FUNCTION_BLOCK  FB_NCU_Base
//////////////////
// NCU Function 
//////////////////
VAR_INPUT PERSISTENT
	// Parameters of the Object (instance/model specific) 
	ParamIPAddress				: STRING := '192.168.1.1' ; // IP 
	ParamTcpPort				: UINT		:= 502;
	ParamTimeOut				: TIME := T#10S ; 
	ParamClockReadTime			: TIME := T#1S ; 
	
	ParamClockWriteTime			: TIME := T#1S ; 	
	
	ParamUnitID 				: BYTE:=1; 					// (NA)   SMA Modbus Unit ID.
	ParamNbTracker				: BYTE ; 					// Number of tracker behind the 
	ParamNCUNum					: INT ; 					// Numerous of TCU 
	                                                		
	ParamTempoComAlarm			: TIME 			 ; 			// (s) Config : Tempo to detect LOC Alarm	

END_VAR

VAR_INPUT 
	//Child objects
	IN_CmdReset_L							: BOOL;				// (NA) External Reset Command	
    IN_CmdToggleRead						: BOOL;
    IN_CmdToggleWrite						: BOOL;
END_VAR


VAR
	//M_ROTATE VARIABLES//
	
		
	//M_ALARMMANAGEMENT VARIABLES//
		TON_ComAlarm				: TON ; 												// Tempo before detecting loss of communication. 
	
	
		
	//M_READ VARAIBLES 
	
		
	//M_STATEMANAGER VARIABLES//
	
		
	// M_EXECUTE VARIABLES 	//      
		TP1							: TP ; 				// (NA) Tempo to define Modbus Reading Frequency 
		TP2 						: TP ; 				// (NA) Tempo to define Modbus Writing Frequency
		                            
		ClockRead					: BOOL;				// (NA) Modbus reading Clock
		ClockWrite 					: BOOL;				// (NA) Modbus writing Clock 	

    //M_CP VARIABLES//
		Trig_Cmd_Read						: R_TRIG;                                                                                        
		Trig_Cmd_Write						: R_TRIG;                                                                                        
	//M_INIT VARIABLES // 	        		
		bInit								: BOOL := TRUE ; 		// (NA) Initialize object parameters at first cycle 
				
END_VAR

METHOD M_AlarmManagement
//////////////////
// Manages Contactor alarms and warnings
/////////////////

VAR 
	// Method local variables (reinitialized at each cycle) 
	
END_VAR
END_METHOD

METHOD M_CP 
VAR_INPUT
END_VAR
END_METHOD

METHOD M_Execute
VAR_INPUT
END_VAR

VAR

END_VAR




// READING AND WRITING CLOCK //
	TP1(IN:=NOT TP1.Q , PT:= ParamClockReadTime);
	ClockRead 				:= TP1.Q;

	TP2(IN:=NOT TP2.Q , PT:= ParamClockWriteTime);
	ClockWrite 				:= TP2.Q;

// PERMANENT CONDITIONS //	
	
	
//Methods call	
	M_Read();
	M_Rotate(); 

	M_AlarmManagement();
END_METHOD

METHOD M_Read
//////////////////
// Manages Opening of the contactor
//////////////////

VAR 
	// Method local variables (reinitialized at each cycle) 
	KK: WORD ; 
	LL: WORD ; 
	JJ: WORD;
	MW: FB_MergeWordsToDint;
	MF : FB_MergeWordsToFloat ; 

	MesFlag				: ARRAY[1..5] OF  WORD;	
	MesAlarm2			: ARRAY[1..5] OF WORD;
	MesAlarm			: ARRAY[1..5] OF WORD;
	MesStatus			: ARRAY[1..5] OF WORD ; 
	MesStatusSynthesis	: WORD ; 

	CalTraNb: UINT;
END_VAR
END_METHOD

METHOD M_Rotate
//////////////////
// Manages Opening of the contactor
//////////////////

VAR 
	// Method local variables (reinitialized at each cycle) 

	CHECK: BOOL ;
	WriteCmd: BOOL ;
	CHECK1: BOOL ;
	WriteCmd1: BOOL ;	
	CHECK2: BOOL ;
	WriteCmd2: BOOL ;	
	CHECK3: BOOL ;
	WriteCmd3: BOOL ;	
		
	
	SetptGroupCmd		: WORD ; 




	FRS1: BOOL;

END_VAR
END_METHOD

END_FUNCTION_BLOCK

(* stored: Version 1.1.0.1
   POU FB_NCU_Base: Id {e070f539-9f0f-4afd-ad1d-5c738321e762}, SpecialFunc None
   Method M_AlarmManagement: Id {45f68959-3abf-4272-a977-c973f8a127a9}
   Method M_CP: Id {abf456c9-672c-4781-a1ed-8c2e426120e9}
   Method M_Execute: Id {31bc01cf-6276-428e-81dd-8eb67265daae}
   Method M_Read: Id {8ae70366-d19c-4383-8dda-5eb0b93c28af}
   Method M_Rotate: Id {92e25784-f75a-4d4d-adf9-38e890c36ca3} *)
